Omron CX-Programmer project NewProject (CX-Programmer 9.75)

# PLC PARKING_PROJECT: CJ2M CPU11

## Global symbols (name address type ; comment)
0.01 BOOL  ; S1
0.02 BOOL  ; S2
0.03 BOOL  ; DUMMY BABA
100.00 BOOL  ; IN OPEN
100.01 BOOL  ; IN CLOSE
100.02 BOOL  ; OUT OPEN
100.03 BOOL  ; OUT CLOSE
T0000 BOOL  ; T0
T0001 BOOL  ; T1

## Program NewProgram1 (cyclic task 0)
Local symbols
NOT BOOL

### Section Section1

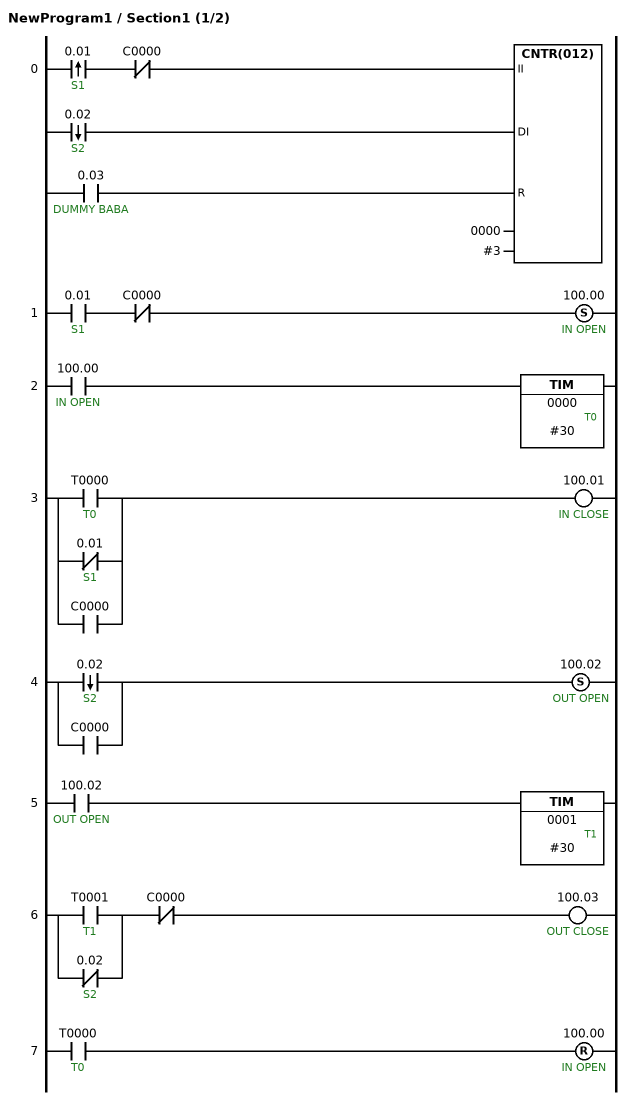
; rung 0
@LD 0.01  ; S1
ANDNOT C0000
%LD 0.02  ; S2
LD 0.03  ; DUMMY BABA
CNTR(012) 0000 #3
; rung 1
LD 0.01  ; S1
ANDNOT C0000
SET 100.00  ; IN OPEN
; rung 2
LD 100.00  ; IN OPEN
TIM 0000 #30  ; T0
; rung 3
LD T0000  ; T0
ORNOT 0.01  ; S1
OR C0000
OUT 100.01  ; IN CLOSE
; rung 4
%LD 0.02  ; S2
OR C0000
SET 100.02  ; OUT OPEN
; rung 5
LD 100.02  ; OUT OPEN
TIM 0001 #30  ; T1
; rung 6
LD T0001  ; T1
ORNOT 0.02  ; S2
ANDNOT C0000
OUT 100.03  ; OUT CLOSE
; rung 7
LD T0000  ; T0
RSET 100.00  ; IN OPEN

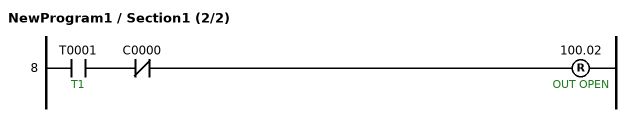
; rung 8
LD T0001  ; T1
ANDNOT C0000
RSET 100.02  ; OUT OPEN

### Section END
; rung 0
END(001)